# B&R Automation Studio project VisionSample (part 5)

#### Main.st
```iecst
// --------------------------------------------------------------------------------------------------------------------
// This task calculates the nettime depending on a drive velocity
// - This task must run at the same cycle as the Powerlink bus
// - Make sure that nettime is selected in the vision application (Image aquisition -> Aquisition configuration -> Trigger Source -> Trigger delay
// --------------------------------------------------------------------------------------------------------------------
PROGRAM _INIT
	gVisionNettime.CMD.Activate					:= TRUE;
	gVisionNettime.CFG.AxisPeriod				:= 360; // Needs also to be set in the axis configuration
	gVisionNettime.CFG.AxisPositionTrigger		:= 0;
	gVisionNettime.CFG.AxisPositionDelay_Cycles	:= 1; 	// Number of PLK cycles which the axis position is old when it comes to this task (Time from encoder to now in this task)
	gVisionNettime.CFG.VisionPreTrigger_Cycles	:= 4; 	// Number of powerlink cycles the trigger has to be send ahead
														// For camera only 4 is good value, for backlight use 12 with a 800us Powerlink cylce
END_PROGRAM

// -----------------------------------------------------------------------------------------------------------
// Cyclic part
// -----------------------------------------------------------------------------------------------------------
PROGRAM _CYCLIC
	PowerlinkCycle_us			:= NettimeCurrent_us - NettimeLastCycle_us;
	NettimeLastCycle_us			:= NettimeCurrent_us;
	IF gVisionNettime.CMD.Activate AND gVisionNettime.DAT.AxisInVelocity AND gVisionNettime.DAT.AxisVelocity > 0 THEN
		AxisPositionNow			:= gVisionNettime.DAT.AxisPosition + gVisionNettime.DAT.AxisVelocity * PowerlinkCycle_us * gVisionNettime.CFG.AxisPositionDelay_Cycles / 1000000; // When the MpAxis gives us the read position, it is old. So calculate the "now" position
		IF AxisPositionNow > gVisionNettime.CFG.AxisPeriod THEN // modulo correction
			AxisPositionNow		:= AxisPositionNow - gVisionNettime.CFG.AxisPeriod;
		ELSIF AxisPositionNow < 0 THEN // modulo correction
			AxisPositionNow		:= AxisPositionNow + gVisionNettime.CFG.AxisPeriod;
		END_IF
		IF gVisionNettime.DAT.AxisVelocity > 0 THEN
			TriggerPosDelta		:= gVisionNettime.CFG.AxisPositionTrigger - AxisPositionNow;
		ELSE
			TriggerPosDelta		:= AxisPositionNow - gVisionNettime.CFG.AxisPositionTrigger;
		END_IF
		IF TriggerPosDelta < 0 THEN // modulo correction
			TriggerPosDelta		:= TriggerPosDelta + gVisionNettime.CFG.AxisPeriod;
		END_IF
		TriggerTimeDelta_us := LREAL_TO_DINT((TriggerPosDelta / gVisionNettime.DAT.AxisVelocity) * 1000000);
		// Wait for the moment that axis is in the send trigger window depend on delay by topology and the actual powerlink cycle
		IF (TriggerTimeDelta_us >= (gVisionNettime.CFG.VisionPreTrigger_Cycles)     * PowerlinkCycle_us) AND
		   (TriggerTimeDelta_us <= (gVisionNettime.CFG.VisionPreTrigger_Cycles + 1) * PowerlinkCycle_us) THEN
			gVisionNettime.DAT.NettimeNext_us	:= NettimeCurrent_us + TriggerTimeDelta_us;
			gVisionNettime.DAT.NettimeDelta_us	:= TriggerTimeDelta_us;
			// Transfer nettime to sensor and fire trigger
			IF gVisionSensor[gSelectedSensor].HW.Ready AND NOT gVisionSensor[gSelectedSensor].DAT.ImageProcessingActive THEN
				gVisionSensor[gSelectedSensor].CMD.ImageTrigger	:= TRUE;
				gVisionSensor[gSelectedSensor].DAT.NettimeDelay	:= gVisionNettime.DAT.NettimeNext_us;
			ELSE
				gVisionNettime.DAT.Overflow := gVisionNettime.DAT.Overflow + 1;
			END_IF
		END_IF
	END_IF
END_PROGRAM
```

### Program Logical/Vision/Axis (IEC)

#### Main.st - Init, cyclic, exit code
```iecst
// --------------------------------------------------------------------------------------------------------------------
// Motion sample for using nettime
// --------------------------------------------------------------------------------------------------------------------
PROGRAM _INIT
	MpAxisBasic_0.Enable			:= TRUE;
	MpAxisBasic_0.MpLink			:= ADR(gAxis_1);
	MpAxisBasic_0.Parameters		:= ADR(MpAxisBasicPar_0);
	MpAxisBasic_0();
	MpAxisBasicPar_0.Homing.Mode	:= mcHOMING_DEFAULT;
END_PROGRAM

// -----------------------------------------------------------------------------------------------------------
// Cyclic part
// -----------------------------------------------------------------------------------------------------------
PROGRAM _CYCLIC
	MpAxisBasic_0.Power					:= MpAxisBasic_0.Active AND MpAxisBasic_0.Info.ReadyToPowerOn AND cmdAxisPower;
	MpAxisBasic_0.ErrorReset			:= cmdAxisErrorReset;
	MpAxisBasic_0.Home					:= MpAxisBasic_0.PowerOn AND NOT MpAxisBasic_0.IsHomed XOR cmdAxisHome;
	MpAxisBasic_0.MoveVelocity			:= MpAxisBasic_0.PowerOn AND MpAxisBasic_0.IsHomed AND cmdAxisRun;
	IF MpAxisBasic_0.PowerOn AND MpAxisBasic_0.IsHomed AND cmdAxisMoveAbs THEN
		MpAxisBasic_0.MoveAbsolute		:= TRUE;
		MpAxisBasicPar_0.Position		:= gVisionNettime.CFG.AxisPositionTrigger;
	END_IF
	cmdAxisMoveAbs					:= FALSE;
	IF AxisVelocity <> MpAxisBasicPar_0.Velocity OR AxisAcceleration <> MpAxisBasicPar_0.Acceleration THEN
		MpAxisBasicPar_0.Velocity		:= AxisVelocity;
		MpAxisBasicPar_0.Acceleration	:= AxisAcceleration;
		MpAxisBasicPar_0.Deceleration	:= AxisAcceleration;
		MpAxisBasic_0.Update			:= TRUE;
	END_IF
	MpAxisBasic_0();
	gVisionNettime.DAT.AxisInVelocity	:= MpAxisBasic_0.InVelocity;
	gVisionNettime.DAT.AxisPosition		:= MpAxisBasic_0.Position;
	gVisionNettime.DAT.AxisVelocity		:= MpAxisBasic_0.Velocity;
	IF MpAxisBasic_0.UpdateDone THEN
		MpAxisBasic_0.Update := FALSE;
	END_IF
	IF MpAxisBasic_0.InPosition THEN
		MpAxisBasic_0.MoveAbsolute		:= FALSE;
	END_IF
END_PROGRAM
```

#### Variables.var - Local variables
```iecst
VAR
	MpAxisBasicPar_0 : MpAxisBasicParType; (*Motion parameters*)
	MpAxisBasic_0 : MpAxisBasic; (*Basic motion function block*)
	AxisVelocity : REAL := 360; (*Velocity for movement*)
	AxisAcceleration : REAL := 36000; (*Acceleration and deceleration for movement*)
	cmdAxisRun : BOOL;
	cmdAxisPower : BOOL;
	cmdAxisHome : BOOL;
	cmdAxisMoveAbs : BOOL;
	cmdAxisErrorReset : BOOL;
END_VAR
```

#### gAxisTypes.typ - not listed in the package file held
```iecst
(*-----------------------------------------------------------------------------------------------------------------------------------------*)
(*General vision structures*)

TYPE
	gAxis_status_typ : 	STRUCT
		position : REAL;
		velocity : REAL;
		inVelocity : BOOL;
		triggerTimeDelta : DINT;
		nettime : DINT;
		powerlinkCycleTime : DINT;
	END_STRUCT;
	gAxis_typ : 	STRUCT
		status : gAxis_status_typ;
	END_STRUCT;
END_TYPE
```

#### gAxis.var - not listed in the package file held
```iecst
VAR
	gAxis : gAxis_typ;
END_VAR
```

#### Program Logical/Vision/Axis/Axis

##### Variables.var
```iecst
VAR
	this : local_typ;
	hw : hw_typ;
	hmi : hmi_typ;
END_VAR
```

##### Main.st
```iecst
// --------------------------------------------------------------------------------------------------------------------
// Motion sample for using nettime
// --------------------------------------------------------------------------------------------------------------------
PROGRAM _INIT
	this.mpAxisBasic_0.Enable			:= TRUE;
	this.mpAxisBasic_0.MpLink			:= ADR(gAxis_1);
	this.mpAxisBasic_0.Parameters		:= ADR(this.mpAxisBasicPar_0);
	this.mpAxisBasic_0();
	this.mpAxisBasicPar_0.Homing.Mode	:= mcHOMING_DEFAULT;

	gVisionNettime.CMD.Activate					:= TRUE;
	hmi.in.recipe.axisPeriod				:= 360; // Needs also to be set in the axis configuration
	hmi.in.recipe.axisPositionTrigger		:= 0;
	hmi.in.recipe.axisPositionDelayCycles	:= 1; 	// Number of PLK cycles which the axis position is old when it comes to this task (Time from encoder to now in this task)
	hmi.in.recipe.visionPreTriggerCycles	:= 4; 	// Number of powerlink cycles the trigger has to be send ahead
	// For camera only 4 is good value, for backlight use 12 with a 800us Powerlink cylce

END_PROGRAM

// -----------------------------------------------------------------------------------------------------------
// Cyclic part
// -----------------------------------------------------------------------------------------------------------
PROGRAM _CYCLIC

// -----------------------------------------------------------------------------------------------------------
// Mapp Motion Axis control
// -----------------------------------------------------------------------------------------------------------
	this.mpAxisBasic_0.Power				:= this.mpAxisBasic_0.Active AND this.mpAxisBasic_0.Info.ReadyToPowerOn AND hmi.in.cmd.power;
	this.mpAxisBasic_0.ErrorReset			:= hmi.in.cmd.errReset;
	this.mpAxisBasic_0.Home					:= this.mpAxisBasic_0.PowerOn AND NOT this.mpAxisBasic_0.IsHomed XOR hmi.in.cmd.home;
	this.mpAxisBasic_0.MoveVelocity			:= this.mpAxisBasic_0.PowerOn AND this.mpAxisBasic_0.IsHomed AND hmi.in.cmd.run;

	IF this.mpAxisBasic_0.PowerOn AND this.mpAxisBasic_0.IsHomed AND hmi.in.cmd.moveAbs THEN
		this.mpAxisBasic_0.MoveAbsolute		:= TRUE;
		this.mpAxisBasicPar_0.Position		:= gVisionNettime.CFG.AxisPositionTrigger;
	END_IF
	hmi.in.cmd.moveAbs					:= FALSE;

	IF hmi.in.recipe.velocity <> this.mpAxisBasicPar_0.Velocity OR hmi.in.recipe.acceleration <> this.mpAxisBasicPar_0.Acceleration THEN
		this.mpAxisBasicPar_0.Velocity		:= hmi.in.recipe.velocity;
		this.mpAxisBasicPar_0.Acceleration	:= hmi.in.recipe.acceleration;
		this.mpAxisBasicPar_0.Deceleration	:= hmi.in.recipe.acceleration;
		this.mpAxisBasic_0.Update			:= TRUE;
	END_IF

	this.mpAxisBasic_0();

	IF hw.in.nettime > this.nettimeLastCycle_us THEN
		this.powerlinkCycle_us	:= hw.in.nettime - this.nettimeLastCycle_us;
	ELSE
		this.powerlinkCycle_us	:= -2147483648-hw.in.nettime + 2147483647-this.nettimeLastCycle_us; // handle wrap around
	END_IF
	this.nettimeLastCycle_us		:= hw.in.nettime;

	hmi.out.inVelocity 	:= gAxis.status.inVelocity	:= 	this.mpAxisBasic_0.InVelocity;
	hmi.out.veleocity 	:= gAxis.status.velocity	:= 	this.mpAxisBasic_0.Velocity;
	hmi.out.inPostion 								:=	this.mpAxisBasic_0.InPosition;
	// When the MpAxis gives us the read position, it is old. So calculate the "now" position
	hmi.out.positon 	:= gAxis.status.position	:= 	LREAL_TO_REAL(this.mpAxisBasic_0.Position) + this.mpAxisBasic_0.Velocity * DINT_TO_REAL(this.powerlinkCycle_us) * hmi.in.recipe.axisPositionDelayCycles / 1000000; ;

	IF this.mpAxisBasic_0.UpdateDone THEN
		this.mpAxisBasic_0.Update := FALSE;
	END_IF

	IF this.mpAxisBasic_0.InPosition THEN
		this.mpAxisBasic_0.MoveAbsolute		:= FALSE;
	END_IF

	// -----------------------------------------------------------------------------------------------------------
	// Calulate time to camera trigger point
	// -----------------------------------------------------------------------------------------------------------

	// calculate axis postion in the current period
	IF this.axisPositionNow > hmi.in.recipe.axisPeriod THEN // modulo correction
		this.axisPositionNow		:= hmi.out.positon- hmi.in.recipe.axisPeriod;
	ELSIF this.axisPositionNow < 0 THEN // modulo correction
		this.axisPositionNow		:= hmi.out.positon + hmi.in.recipe.axisPeriod;
	END_IF

	// calculate differen (triggerPosDelta) in current axis postion to the trigger postion
	IF this.mpAxisBasic_0.Velocity > 0 THEN
		this.triggerPosDelta		:= hmi.in.recipe.axisPositionTrigger - this.axisPositionNow;
	ELSE
		this.triggerPosDelta		:= this.axisPositionNow - hmi.in.recipe.axisPositionTrigger;
	END_IF

	IF this.triggerPosDelta < 0 THEN // modulo correction
		this.triggerPosDelta		:= this.triggerPosDelta + hmi.in.recipe.axisPositionTrigger;
	END_IF

	IF hmi.out.veleocity > 0 THEN
		// convert position difference to a time difference (the time until the axis is at the trigger postion with the current velocity)
		gAxis.status.triggerTimeDelta 	:= LREAL_TO_DINT((this.triggerPosDelta / this.mpAxisBasic_0.Velocity) * 1000000);
	END_IF

	gAxis.status.nettime 		  		:= hw.in.nettime;
	gAxis.status.powerlinkCycleTime 	:= this.powerlinkCycle_us;

	hmi.out.triggerPosDelta 	:= this.triggerPosDelta;
	hmi.out.powerlinkCycle_us 	:= this.powerlinkCycle_us;
	hmi.out.triggerTimeDelta 	:= this.triggerTimeDelta;

END_PROGRAM
```

### Program Logical/Vision/YourTask (IEC)

#### Types.typ
```iecst
TYPE
	enumViMotion :
		(
		stINIT,
		stPOWER,
		stHOME,
		stREADY,
		stRUN
		);
END_TYPE
```

#### Main.st
```iecst
// -----------------------------------------------------------------------------------------------------------
// Use this task to add your own code
// -----------------------------------------------------------------------------------------------------------

// -----------------------------------------------------------------------------------------------------------
// Initialization
// -----------------------------------------------------------------------------------------------------------
PROGRAM _INIT
END_PROGRAM

// -----------------------------------------------------------------------------------------------------------
// Cyclic part
// -----------------------------------------------------------------------------------------------------------
PROGRAM _CYCLIC
	// -----------------------------------------------------------------------------------------------------------
	// Vision sensor configuration
	// -----------------------------------------------------------------------------------------------------------
	// Configuration for blob
	gVisionSensor[1].CFG.VisionFunction		:= enumBlob;			// Used to run specific code for this vision function
	gVisionSensor[1].CFG.PowerlinkNode		:= 1;					// Powerlink node number
	gVisionSensor[1].CFG.DataStructure		:= ADR(gBlob);			// Global structures that holds all data related to this function
	gVisionSensor[1].CFG.ComponentLink		:= gCameraBlob;			// Vision component name defined under mappVision in the configuration view
	gVisionSensor[1].CFG.ResolutionWidth	:= 1280;
	gVisionSensor[1].CFG.ResolutionHeight	:= 1024;
	// Configuration for code reader
	gVisionSensor[2].CFG.VisionFunction		:= enumCoderReader;
	gVisionSensor[2].CFG.PowerlinkNode		:= 2;
	gVisionSensor[2].CFG.DataStructure		:= ADR(gCodeReader);
	gVisionSensor[2].CFG.ComponentLink		:= gCameraCodeReading;
	gVisionSensor[2].CFG.ResolutionWidth	:= 1280;
	gVisionSensor[2].CFG.ResolutionHeight	:= 1024;
	// Configuration for match
	gVisionSensor[3].CFG.VisionFunction		:= enumMatch;
	gVisionSensor[3].CFG.PowerlinkNode		:= 3;
	gVisionSensor[3].CFG.DataStructure		:= ADR(gMatch);
	gVisionSensor[3].CFG.ComponentLink		:= gCameraMatch;
	gVisionSensor[3].CFG.ResolutionWidth	:= 1280;
	gVisionSensor[3].CFG.ResolutionHeight	:= 1024;
	// Configuration for meaurement
	gVisionSensor[4].CFG.VisionFunction		:= enumMeasurement;
	gVisionSensor[4].CFG.PowerlinkNode		:= 4;
	gVisionSensor[4].CFG.DataStructure		:= ADR(gMT);
	gVisionSensor[4].CFG.ComponentLink		:= gCameraMeasurement;
	gVisionSensor[4].CFG.ResolutionWidth	:= 1280;
	gVisionSensor[4].CFG.ResolutionHeight	:= 1024;
	// Configuration for OCR
	gVisionSensor[5].CFG.VisionFunction		:= enumOCR;
	gVisionSensor[5].CFG.PowerlinkNode		:= 5;
	gVisionSensor[5].CFG.DataStructure		:= ADR(gOCR);
	gVisionSensor[5].CFG.ComponentLink		:= gCameraOCR;
	gVisionSensor[5].CFG.ResolutionWidth	:= 1280;
	gVisionSensor[5].CFG.ResolutionHeight	:= 1024;
	// Configuration for PixelCounter
	gVisionSensor[6].CFG.VisionFunction		:= enumPixelCounter;
	gVisionSensor[6].CFG.PowerlinkNode		:= 6;
	gVisionSensor[6].CFG.DataStructure		:= ADR(gPixel);
	gVisionSensor[6].CFG.ComponentLink		:= gCameraPxl;
	gVisionSensor[6].CFG.ResolutionWidth	:= 1280;
	gVisionSensor[6].CFG.ResolutionHeight	:= 1024;

	// -----------------------------------------------------------------------------------------------------------
	// Lights configuration
	// -----------------------------------------------------------------------------------------------------------
	// Configuration for backlights
	gVisionLight[1].CFG.LightType		:= enumBacklight;
	gVisionLight[1].CFG.PowerlinkNode	:= 10;
	gVisionLight[1].DAT.FlashColor		:= 1;
	gVisionLight[2].CFG.LightType		:= enumBacklight;
	gVisionLight[2].CFG.PowerlinkNode	:= 11;
	gVisionLight[2].DAT.FlashColor		:= 1;
	// Configuration for lightbars
	gVisionLight[3].CFG.LightType		:= enumLightbar;
	gVisionLight[3].CFG.PowerlinkNode	:= 20;
	gVisionLight[3].DAT.FlashColor		:= 1;

	// -----------------------------------------------------------------------------------------------------------
	// Backlight handling, this block can be deleted when no backlights are used
	// -----------------------------------------------------------------------------------------------------------

	// -----------------------------------------------------------------------------------------------------------
	// Trigger selected backlight when selected sensor is triggered
	IF(EDGEPOS(gVisionSensor[gSelectedSensor].CMD.ImageTrigger)) THEN
		gVisionLight[gSelectedLight].DAT.Exposure		:= gVisionSensor[gSelectedSensor].DAT.Exposure;
		gVisionLight[gSelectedLight].DAT.NettimeDelay	:= gVisionSensor[gSelectedSensor].DAT.NettimeDelay;
		gVisionLight[gSelectedLight].CMD.FlashTrigger	:= TRUE;
	END_IF

END_PROGRAM
```

### gFiles.typ
```iecst
TYPE
	gFiles_output_typ : 	STRUCT
		fileDevice : STRING[10];
		ready : BOOL;
	END_STRUCT;
	gFiles_typ : 	STRUCT
		output : gFiles_output_typ;
	END_STRUCT;
END_TYPE
```

### gFiles.var
```iecst
VAR
	gFiles : gFiles_typ;
END_VAR
```

### Program Logical/Vision/Files/Files (IEC)

#### Types.typ
```iecst
TYPE
	local_typ : 	STRUCT
		brdkFileDevUsb : brdkFileDeviceHandler;
		brdkFileDev : brdkFileDeviceHandler;
	END_STRUCT;
END_TYPE
```

#### Variables.var
```iecst
VAR
	this : local_typ;
END_VAR
```

#### Main.st
```iecst
PROGRAM _INIT
	(* Insert code here *)
	this.brdkFileDev.enable := TRUE;
	this.brdkFileDev.setup.plcDrive := F_DRIVE;
	this.brdkFileDev.setup.usbOverrule := FALSE;
	this.brdkFileDev.simulation.pcRootFolder := 'plcSim\MappVisionDemo';
	this.brdkFileDev.simulation.pcHDDrive := C_DRIVE;
	this.brdkFileDev.setup.rootFileDeviceName := 'ROOT_PLC';

	this.brdkFileDev.setup.fileDevices[0].name := 'SIM_BLOB';
	this.brdkFileDev.setup.fileDevices[0].path := 'sim/BLOB';
	this.brdkFileDev.setup.fileDevices[1].name := 'SIM_CR';
	this.brdkFileDev.setup.fileDevices[1].path := 'sim/CR';
	this.brdkFileDev.setup.fileDevices[2].name := 'SIM_MATCH';
	this.brdkFileDev.setup.fileDevices[2].path := 'sim/Match';
	this.brdkFileDev.setup.fileDevices[3].name := 'SIM_MEAS';
	this.brdkFileDev.setup.fileDevices[3].path := 'sim/Measurement';
	this.brdkFileDev.setup.fileDevices[4].name := 'SIM_OCR';
	this.brdkFileDev.setup.fileDevices[4].path := 'sim/OCR';
	this.brdkFileDev.setup.fileDevices[5].name := 'SIM_PXCNT';
	this.brdkFileDev.setup.fileDevices[5].path := 'sim/PxCnt';

	this.brdkFileDevUsb.setup.plcDrive := F_DRIVE;
	this.brdkFileDevUsb.setup.usbOverrule := TRUE;
	this.brdkFileDevUsb.simulation.pcRootFolder := 'plcSim\MappVisionDemo';
	this.brdkFileDevUsb.simulation.pcHDDrive := C_DRIVE;
	this.brdkFileDevUsb.simulation.pcUSBDrive := D_DRIVE;
	this.brdkFileDevUsb.setup.rootFileDeviceName := 'ROOT_USB';

	this.brdkFileDevUsb.setup.fileDevices[0].name := 'IMG';
	this.brdkFileDevUsb.setup.fileDevices[0].path := 'images';
	this.brdkFileDevUsb.setup.fileDevices[1].name := 'RECIPE';
	this.brdkFileDevUsb.setup.fileDevices[1].path := 'Recipe';
	this.brdkFileDevUsb.setup.fileDevices[2].name := 'VI_DIAG';
	this.brdkFileDevUsb.setup.fileDevices[2].path := 'visionDiag';

END_PROGRAM

PROGRAM _CYCLIC
	(* Insert code here *)

	this.brdkFileDev();

	IF EDGEPOS(this.brdkFileDev.ready) THEN
		this.brdkFileDevUsb.enable := TRUE;
	END_IF

	this.brdkFileDevUsb();

	gFiles.output.fileDevice := 'ROOT';
	gFiles.output.ready := this.brdkFileDevUsb.ready;

END_PROGRAM

PROGRAM _EXIT
	(* Insert code here *)

	END_PROGRAM
```

### Program Logical/Vision/Vi_Color (IEC)

#### Main.st - Init, cyclic, exit code
```iecst
PROGRAM _INIT
	// ---------------------------------------------------------------------------------------------------------------------
	// Camera configuration
	gVisionSensor[VI_COLOR_SENSOR].DAT.Gain := 1;
	gVisionSensor[VI_COLOR_SENSOR].DAT.Focus := 14000;
	gVisionSensor[VI_COLOR_SENSOR].DAT.Exposure := 150;
	gVisionSensor[VI_COLOR_SENSOR].DAT.ChromaticLock := TRUE;
	gBlob.EnhancedBlobInformation := TRUE;
	visTableNo;

END_PROGRAM

PROGRAM _CYCLIC
	CASE Step OF
		// ---------------------------------------------------------------------------------------------------------------------
		// Wait for new upload command
		VISTEP_WAIT:
			gVisionColor.DAT.Status := ERR_OK;
			IF gVisionColor.CMD.Evaluate OR gVisionColor.CMD.Teach THEN
				idx := 1;
				brsmemset(ADR(gVisionColor.DAT), 0, SIZEOF(gVisionColor.DAT));
				gVisionColor.CFG.TeachingIndex := visSelectedProduct + 1;
				gVisionColor.DAT.Status := ERR_FUB_BUSY;
				gVisionSensor[VI_COLOR_SENSOR].DAT.Enable := TRUE;
				Step := VISTEP_FLASH;
			END_IF
			// ---------------------------------------------------------------------------------------------------------------------
			// Teach new color
		VISTEP_FLASH:
			// Flash with all available colors
			IF(idx = 1 AND gVisionColor.CFG.FlashColor1 <> 0) THEN
				gVisionSensor[VI_COLOR_SENSOR].DAT.FlashColor := gVisionColor.CFG.FlashColor1;
			ELSIF(idx = 2 AND gVisionColor.CFG.FlashColor2 <> 0) THEN
				gVisionSensor[VI_COLOR_SENSOR].DAT.FlashColor := gVisionColor.CFG.FlashColor2;
			ELSIF(idx = 3 AND gVisionColor.CFG.FlashColor3 <> 0) THEN
				gVisionSensor[VI_COLOR_SENSOR].DAT.FlashColor := gVisionColor.CFG.FlashColor3;
			ELSIF(idx = 4 AND gVisionColor.CFG.FlashColor4 <> 0) THEN
				gVisionSensor[VI_COLOR_SENSOR].DAT.FlashColor := gVisionColor.CFG.FlashColor4;
				// Finish flashing when no color is set
			ELSE
				IF(gVisionColor.CMD.Teach) THEN
					gVisionColor.CMD.Teach := FALSE;
					Step := VISTEP_WAIT;
				ELSE
					Step := VISTEP_CHECK;
				END_IF
				RETURN;
			END_IF
			// Take new image with selected color
			IF NETTIME_ENABLE THEN
				gVisionSensor[VI_COLOR_SENSOR].DAT.NettimeDelay := NettimeCurrent_us + NETTIME_DEFAULT_DELAY;
			END_IF
			gVisionSensor[VI_COLOR_SENSOR].CMD.ImageTrigger 	:= TRUE;
			IF(gVisionColor.CMD.Teach) THEN
				Step := VISTEP_TEACH;
			ELSE
				Step := VISTEP_CHECK;
			END_IF
			// ---------------------------------------------------------------------------------------------------------------------
			// Teach new color
		VISTEP_TEACH:
			// Wait for trigger to finish
			IF(gVisionSensor[VI_COLOR_SENSOR].CMD.ImageTrigger = FALSE) THEN
				IF(gVisionSensor[VI_COLOR_SENSOR].DAT.ResultCnt > 0)  THEN
					IF(idx = 1) THEN
						gVisionColor.CFG.GrayValue1[gVisionColor.CFG.TeachingIndex] := gBlob.MeanGrayValue[1];
					ELSIF(idx = 2) THEN
						gVisionColor.CFG.GrayValue2[gVisionColor.CFG.TeachingIndex] := gBlob.MeanGrayValue[1];
					ELSIF(idx = 3) THEN
						gVisionColor.CFG.GrayValue3[gVisionColor.CFG.TeachingIndex] := gBlob.MeanGrayValue[1];
					ELSIF(idx = 4) THEN
						gVisionColor.CFG.GrayValue4[gVisionColor.CFG.TeachingIndex] := gBlob.MeanGrayValue[1];
					END_IF
					//
					idx := idx + 1;
					IF(idx > 4) THEN
						gVisionColor.CMD.Teach := FALSE;
						Step := VISTEP_WAIT;
					ELSE
						Step := VISTEP_FLASH;
					END_IF
				ELSE
					gVisionColor.DAT.Status := ERR_VI_COLOR_IDENTIFY;
					Step := VISTEP_ERR;
				END_IF
			END_IF
			// ---------------------------------------------------------------------------------------------------------------------
			// Check new product
		VISTEP_CHECK:
			// Wait for trigger to finish
			IF(gVisionSensor[VI_COLOR_SENSOR].CMD.ImageTrigger = FALSE) THEN
				IF(gVisionSensor[VI_COLOR_SENSOR].DAT.ResultCnt > 0)  THEN
					IF(idx = 1) THEN
						gVisionColor.DAT.GrayValue1 := gBlob.MeanGrayValue[1];
					ELSIF(idx = 2) THEN
						gVisionColor.DAT.GrayValue2 := gBlob.MeanGrayValue[1];
					ELSIF(idx = 3) THEN
						gVisionColor.DAT.GrayValue3 := gBlob.MeanGrayValue[1];
					ELSIF(idx = 4) THEN
						gVisionColor.DAT.GrayValue4 := gBlob.MeanGrayValue[1];
					END_IF
					//
					idx := idx + 1;
					IF(idx > 4) THEN
						gVisionColor.DAT.LowError := 16#FFFF;
						gVisionColor.DAT.LowIndex := 16#FFFF;
						gVisionColor.DAT.LowDistance := 16#FFFF;
						Step := VISTEP_EVAL;
					ELSE
						Step := VISTEP_FLASH;
					END_IF
				ELSE
					gVisionColor.DAT.Status := ERR_VI_COLOR_IDENTIFY;
					Step := VISTEP_ERR;
				END_IF
			END_IF
			// ---------------------------------------------------------------------------------------------------------------------
			// Check new product
		VISTEP_EVAL:
			FOR idx:= 1 TO MAX_NUM_PRODUCTS DO
				// Abort when product gray values are empty
				IF(gVisionColor.CFG.GrayValue1[idx] = 0 AND gVisionColor.CFG.GrayValue2[idx] = 0 AND gVisionColor.CFG.GrayValue3[idx] = 0 AND gVisionColor.CFG.GrayValue4[idx] = 0) THEN
					EXIT;
				END_IF
				// Calculate error for all colors and products
				FOR idy:= 1 TO 4 DO
					IF(idy = 1 AND gVisionColor.CFG.FlashColor1 <> 0) THEN
						gVisionColor.DAT.TotalError[idx] := gVisionColor.DAT.TotalError[idx] + ABS(UINT_TO_INT(gVisionColor.DAT.GrayValue1) - gVisionColor.CFG.GrayValue1[idx]);
					ELSIF(idy = 2 AND gVisionColor.CFG.FlashColor2 <> 0) THEN
						gVisionColor.DAT.TotalError[idx] := gVisionColor.DAT.TotalError[idx] + ABS(UINT_TO_INT(gVisionColor.DAT.GrayValue2) - gVisionColor.CFG.GrayValue2[idx]);
					ELSIF(idy = 3 AND gVisionColor.CFG.FlashColor3 <> 0) THEN
						gVisionColor.DAT.TotalError[idx] := gVisionColor.DAT.TotalError[idx] + ABS(UINT_TO_INT(gVisionColor.DAT.GrayValue3) - gVisionColor.CFG.GrayValue3[idx]);
					ELSIF(idy = 4 AND gVisionColor.CFG.FlashColor4 <> 0) THEN
						gVisionColor.DAT.TotalError[idx] := gVisionColor.DAT.TotalError[idx] + ABS(UINT_TO_INT(gVisionColor.DAT.GrayValue4) - gVisionColor.CFG.GrayValue4[idx]);
					END_IF
				END_FOR;
				// New lowest error
				IF(gVisionColor.DAT.TotalError[idx] < gVisionColor.DAT.LowError) THEN
					gVisionColor.DAT.LowError := gVisionColor.DAT.TotalError[idx];
					gVisionColor.DAT.LowIndex := idx;
					gVisionColor.DAT.LowName := gVisionColor.CFG.ProductName[idx];
				END_IF
			END_FOR;
			// Check distance to next best value
			IF(gVisionColor.DAT.LowIndex <> 16#FFFF) THEN
				FOR idx:= 1 TO MAX_NUM_PRODUCTS DO
					// Abort when product gray values are empty
					IF(gVisionColor.CFG.GrayValue1[idx] = 0 AND gVisionColor.CFG.GrayValue2[idx] = 0 AND gVisionColor.CFG.GrayValue3[idx] = 0 AND gVisionColor.CFG.GrayValue4[idx] = 0) THEN
						EXIT;
					END_IF
					// Store next best product
					IF(gVisionColor.DAT.LowIndex <> idx AND INT_TO_UINT(ABS(UINT_TO_INT(gVisionColor.DAT.TotalError[gVisionColor.DAT.LowIndex])) - gVisionColor.DAT.TotalError[idx]) < gVisionColor.DAT.LowDistance) THEN
						gVisionColor.DAT.LowDistance := ABS(UINT_TO_INT(gVisionColor.DAT.TotalError[gVisionColor.DAT.LowIndex]) - gVisionColor.DAT.TotalError[idx]);
					END_IF
				END_FOR;
				visSelectedProduct := gVisionColor.DAT.LowIndex - 1;
			END_IF
			// Make sure we dont exceed max error
			IF(gVisionColor.DAT.LowError > gVisionColor.CFG.MaxError) THEN
				gVisionColor.DAT.Status := ERR_VI_COLOR_MAX_ERROR;
				Step := VISTEP_ERR;
				// Make sure we have enough distance to next best value
			ELSIF(gVisionColor.DAT.LowDistance < gVisionColor.CFG.MinDifference) THEN
				gVisionColor.DAT.Status := ERR_VI_COLOR_MIN_DISTANCE;
				Step := VISTEP_ERR;
				// Make sure we dont exceed max error
			ELSE
				gVisionColor.CMD.Evaluate := FALSE;
				Step := VISTEP_WAIT;
			END_IF
			// ---------------------------------------------------------------------------------------------------------------------
			// Error state
		VISTEP_ERR:
			IF gVisionColor.CMD.ResetError THEN
				gVisionColor.CMD.ResetError := FALSE;
				gVisionColor.DAT.Status := 0;
				Step := VISTEP_WAIT;
			ELSE
				brsmemset(ADR(gVisionColor.CMD), 0, SIZEOF(gVisionColor.CMD));
			END_IF
	END_CASE
END_PROGRAM
```

#### Variables.var - Local variables
```iecst
(*-----------------------------------------------------------------------------------------------------------------------------------------*)
(*Local variables*)
VAR
	Step : VIStep_Enum;
	idy : UINT;
	idx : UINT;
	visSelectedProduct : UINT;
	visTableNo : ARRAY[1..MAX_NUM_PRODUCTS] OF USINT := [1,2,3,4,5,6,7,8];
END_VAR
(*-----------------------------------------------------------------------------------------------------------------------------------------*)
(*Local constants*)
VAR CONSTANT
	VI_COLOR_SENSOR : USINT := 1; (*Camera index used for color detection*)
END_VAR
(*-----------------------------------------------------------------------------------------------------------------------------------------*)
(*Error contants*)
VAR CONSTANT
	ERR_VI_COLOR_IDENTIFY : UINT := 10000; (*No result found*)
	ERR_VI_COLOR_MAX_ERROR : UINT := 10001; (*Error exceeds maximum value*)
	ERR_VI_COLOR_MIN_DISTANCE : UINT := 10002; (*Next best value is too close*)
END_VAR
```

### Program Logical/Vision/Vi_light

#### Variables.var
```iecst
(*-----------------------------------------------------------------------------------------------------------------------------------------*)
VAR
	VisionLight : REFERENCE TO typLightMain; (*General vision functions that are independent from the inspection function*)
	FlashFailedCntOld : ARRAY[1..MAX_NUM_LIGHTS] OF USINT;
	FlashCompletedCntOld : ARRAY[1..MAX_NUM_LIGHTS] OF USINT;
	visLightsTrigger : BOOL;
	visLightsReset : BOOL;
	visEnableCommand : BOOL;
	visSelectedFlashColor : STRING[10]; (*Flash color string*)
	TriggerTimeout : ARRAY[1..MAX_NUM_LIGHTS] OF TON; (*Disable web reload when timed out*)
	InitialSearchLight : BOOL;
	i : INT;
	visSelectedFlashColorOld : STRING[10];
	visEnableLightBarValues : BOOL;
	idx : UINT;
END_VAR
```

#### Main.st
```iecst
// --------------------------------------------------------------------------------------------------------------------
// General external lights task. This is a support task for the mappView visualization.
// Version 1.x (Check revision history for details)
// --------------------------------------------------------------------------------------------------------------------
PROGRAM _INIT
	// Map global structure to local reference
	VisionLight ACCESS ADR(gVisionLight[visSelectedLight]);

	InitialSearchLight := TRUE;
END_PROGRAM

// -----------------------------------------------------------------------------------------------------------
// Cyclic part
// -----------------------------------------------------------------------------------------------------------
PROGRAM _CYCLIC
// -----------------------------------------------------------------------------------------------------------
// Part 1: Things to be done for every light
// -----------------------------------------------------------------------------------------------------------
	FOR idx := 1 TO MAX_NUM_LIGHTS DO
		// -----------------------------------------------------------------------------------------------------------
		// Reset Light trigger
		// -----------------------------------------------------------------------------------------------------------
		IF (gVisionLight[idx].DAT.FlashCompletedCnt <> FlashCompletedCntOld[idx] OR gVisionLight[idx].DAT.FlashFailedCnt <> FlashFailedCntOld[idx]) THEN
			FlashCompletedCntOld[idx]			:= gVisionLight[idx].DAT.FlashCompletedCnt;
			FlashFailedCntOld[idx]				:= gVisionLight[idx].DAT.FlashFailedCnt;
			gVisionLight[idx].CMD.FlashTrigger	:= FALSE;
		END_IF

		// -----------------------------------------------------------------------------------------------------------
		// Reset trigger when timed out
		// -----------------------------------------------------------------------------------------------------------
		IF gVisionLight[idx].CMD.FlashTrigger THEN
			TriggerTimeout[idx].IN := TRUE;
			TriggerTimeout[idx].PT := REAL_TO_TIME(gVisionLight[idx].DAT.Timeout * 1.25);
			IF TriggerTimeout[idx].Q THEN
				gVisionLight[idx].CMD.FlashTrigger		:= FALSE;
				gVisionLight[idx].CMD.FlashTriggerReset	:= TRUE;
			END_IF
		ELSE
			TriggerTimeout[idx].IN := FALSE;
			gVisionLight[idx].CMD.FlashTriggerReset := FALSE;
		END_IF
		TriggerTimeout[idx]();
	END_FOR

// -----------------------------------------------------------------------------------------------------------
// Part 2: Things to be done for the actual selected light / visualization related things
// -----------------------------------------------------------------------------------------------------------
	// -----------------------------------------------------------------------------------------------------------
	// Select first available light after reboot
	// -----------------------------------------------------------------------------------------------------------
	IF InitialSearchLight THEN
		FOR i := 1 TO MAX_NUM_LIGHTS DO
			IF gVisionLight[i].HW.Connected THEN
				visSelectedLight := i;
				InitialSearchLight := FALSE;
				EXIT;
			END_IF
		END_FOR
	END_IF
	 // -----------------------------------------------------------------------------------------------------------
	// Map global structure to local reference
	// -----------------------------------------------------------------------------------------------------------
	// Make sure we dont exceed array limit
	IF(visSelectedLight > MAX_NUM_LIGHTS) THEN
		visSelectedLight := 1;
	END_IF
	IF(visSelectedLight < 1) THEN
		visSelectedLight := MAX_NUM_LIGHTS;
	END_IF
	VisionLight ACCESS ADR(gVisionLight[visSelectedLight]);

	// -----------------------------------------------------------------------------------------------------------
	// Translate flash color from mappView to IO mapping
	// -----------------------------------------------------------------------------------------------------------
	// Hint: Normally copy from recipe (VisionLight) to visu. Only in case of a change in the visu copy to recipe
	IF visSelectedFlashColor <> visSelectedFlashColorOld THEN // The flash color was changed in the mappView visualization
		VisionLight.DAT.FlashColor := UDINT_TO_USINT(brsatoi(ADR(visSelectedFlashColor)));
	ELSE
		brsitoa(VisionLight.DAT.FlashColor, ADR(visSelectedFlashColor));
	END_IF
	visSelectedFlashColorOld := visSelectedFlashColor;

	// -----------------------------------------------------------------------------------------------------------
	// Reset Light trigger manually
	// -----------------------------------------------------------------------------------------------------------
	IF (visLightsReset) THEN
		VisionLight.CMD.FlashTrigger := FALSE;
		visLightsReset := FALSE;
	END_IF

	// -----------------------------------------------------------------------------------------------------------
	// Fire trigger for lights
	// -----------------------------------------------------------------------------------------------------------
	IF(visLightsTrigger AND VisionLight.HW.Ready) THEN
		// Add default delay and fire trigger
		VisionLight.DAT.NettimeDelay := NettimeCurrent_us + NETTIME_DEFAULT_DELAY;
		VisionLight.CMD.FlashTrigger := TRUE;
		visLightsTrigger := FALSE;
	END_IF

	// -----------------------------------------------------------------------------------------------------------
	// Disable command button when light is disconnected or not ready
	// -----------------------------------------------------------------------------------------------------------
	IF(NOT VisionLight.HW.Connected OR NOT VisionLight.HW.Ready) THEN
		visEnableCommand := FALSE;
	ELSE
		visEnableCommand := TRUE;
	END_IF

	// -----------------------------------------------------------------------------------------------------------
	// Enable fields for different light types
	// -----------------------------------------------------------------------------------------------------------
	visEnableLightBarValues := VisionLight.CFG.LightType = enumLightbar;
END_PROGRAM
```

### Program Logical/Vision/Vi_Optics (IEC)

#### Main.st
```iecst
PROGRAM _INIT

END_PROGRAM
PROGRAM _CYCLIC
	CASE ReadStep OF // Use AsIODiag library to search the ordnernumber of the selcted/plugged camera (eg. VSS112Q22.041P-000) to get the lens and sensor information
		0: // Wait
			IF cmdReadCameraInfo THEN
				cmdReadCameraInfo			:= FALSE;
				Index						:= 0;
				OrderNr						:= '';
				ReadStep := 1;
			END_IF
		1: // Create DiagInformation
			DiagCreateInfo_0.enable			:= TRUE;
			DiagCreateInfo_0.infoKind		:= asdiagPLUGGED;
			DiagCreateInfo_0();
			IF DiagCreateInfo_0.status = 0 THEN
				ReadStep := 2;
			ELSIF DiagCreateInfo_0.status <> ERR_FUB_BUSY THEN
				ReadStep := 90;
			END_IF
		2: // Read HW-ID and compare with selected camera
			DiagGetNumInfo_0.enable			:= TRUE;
			DiagGetNumInfo_0.ident			:= DiagCreateInfo_0.ident;
			DiagGetNumInfo_0.index			:= Index;
			DiagGetNumInfo_0.infoCode		:= asdiagPLUGGED_MODNO;
			DiagGetNumInfo_0();
			IF DiagGetNumInfo_0.status = 0 THEN
				IF DiagGetNumInfo_0.value = gVisionSensor[visSelectedSensor].HW.ID THEN
					ReadStep := 3;
				ELSE
					Index := Index + 1;
					IF Index >= DiagCreateInfo_0.nrEntries THEN
						ReadStep := 91;
					END_IF
				END_IF
			ELSIF DiagGetNumInfo_0.status <> ERR_FUB_BUSY THEN
				ReadStep					:= 92;
			END_IF
		3: // Read ordernumber
			DiagGetStrInfo_0.enable			:= TRUE;
			DiagGetStrInfo_0.ident			:= DiagCreateInfo_0.ident;
			DiagGetStrInfo_0.index			:= Index;
			DiagGetStrInfo_0.infoCode		:= asdiagPLUGGED_MODULE; // Ordnernumber of the plugged module (eg. VSS112Q22.041P-000)
			DiagGetStrInfo_0.pBuffer		:= ADR(OrderNr);
			DiagGetStrInfo_0.bufferLen		:= SIZEOF(OrderNr) - 1;
			DiagGetStrInfo_0();
			IF DiagGetStrInfo_0.status = 0 THEN
				ReadStep := 10;
			ELSIF DiagGetStrInfo_0.status <> ERR_FUB_BUSY THEN
				ReadStep := 93;
			END_IF
		10:
			DiagDisposeInfo_0.enable		:= TRUE;
			DiagDisposeInfo_0.ident			:= DiagCreateInfo_0.ident;
			DiagDisposeInfo_0();
			IF DiagDisposeInfo_0.status = 0 THEN
				ReadStep := 20;
			ELSIF DiagDisposeInfo_0.status <> ERR_FUB_BUSY THEN
				ReadStep := 94;
			END_IF
		20: // get the info to the actual camara, e.g. VSS112Q22.041P-000
			IF brsstrlen(ADR(OrderNr)) = 18 THEN
				pChar ACCESS ADR(OrderNr) + 8; // Letter for Sensor
				CASE pChar OF
					16#31:  Sensor := SENSOR_1_3_MP; // ASCII '1'
					16#32:  Sensor := SENSOR_1_3_MP; // ASCII '2'
					16#34:  Sensor := SENSOR_3_5_MP; // ASCII '4'
					16#35:  Sensor := SENSOR_5_3_MP; // ASCII '5'
				ELSE
					ReadStep := 95;
				END_CASE
				pChar ACCESS ADR(OrderNr) + 10; // first letter for optics (0 or M)
				CASE pChar OF
					16#30:  Lens := LENS_4_6; // ASCII '0'
					16#4D:  Lens := LENS_12_0_MACRO; // ASCII 'M'
				ELSE
					ReadStep := 96;
				END_CASE
				pChar ACCESS ADR(OrderNr) + 11; // second letter for optics
				CASE pChar OF
					16#30:  Lens := LENS_4_6; // ASCII '0' // no optics
					16#32:  Lens := LENS_4_6; // ASCII '2'
					16#33:  Lens := LENS_6_0; // ASCII '3'
					16#34:  Lens := LENS_8_0; // ASCII '4'
					16#35: // ASCII '5'
						IF Lens = LENS_12_0_MACRO THEN
							// do noting, already selected
						ELSE
							Lens := LENS_12_0;
						END_IF
					16#36:  Lens := LENS_16_0; // ASCII '6'
					16#37:  Lens := LENS_25_0; // ASCII '7'
				ELSE
					ReadStep := 97;
				END_CASE
				Distance_mm	:= UINT_TO_LREAL(gVisionSensor[visSelectedSensor].DAT.Focus) / 100.0;
				ReadStep := 0;
			ELSE
				ReadStep := 98;
			END_IF
		90..99: // auto reset errors
			ReadStep := 0;
	END_CASE

	CASE Sensor OF
		SENSOR_1_3_MP:
			PixelSize_um		:= 4.8;
			ResolutionX			:= 1280;
			ResolutionY			:= 1024;
		SENSOR_3_5_MP:
			PixelSize_um		:= 3.2;
			ResolutionX			:= 2112;
			ResolutionY			:= 1664;
		SENSOR_5_3_MP:
			PixelSize_um		:= 3.2;
			ResolutionX			:= 2592;
			ResolutionY			:= 2048;
	END_CASE
	CASE Lens OF
		LENS_4_6:
			FocalLength_mm		:= 4.6;
			MinObjectDist_mm	:= 25;
			MaxObjectDist_mm	:= 65550;
			Aperture			:= 3.5;
		LENS_6_0:
			FocalLength_mm		:= 6.0;
			MinObjectDist_mm	:= 50;
			MaxObjectDist_mm	:= 65550;
			Aperture			:= 3.5;
		LENS_8_0:
			FocalLength_mm		:= 8.0;
			MinObjectDist_mm	:= 50;
			MaxObjectDist_mm	:= 65500;
			Aperture			:= 3.5;
		LENS_12_0:
			FocalLength_mm		:= 12.0;
			MinObjectDist_mm	:= 75;
			MaxObjectDist_mm	:= 5000;
			Aperture			:= 4.0;
		LENS_16_0:
			FocalLength_mm		:= 16.0;
			MinObjectDist_mm	:= 100;
			MaxObjectDist_mm	:= 1500;
			Aperture			:= 4.0;
		LENS_25_0:
			FocalLength_mm		:= 25.0;
			MinObjectDist_mm	:= 250;
			MaxObjectDist_mm	:= 1500;
			Aperture			:= 4.0;
		LENS_12_0_MACRO:
			FocalLength_mm		:= 12.0;
			MinObjectDist_mm	:= 35;
			MaxObjectDist_mm	:= 65;
			Aperture			:= 4.0;
	END_CASE
	ValidDistance					:= Distance_mm >= MinObjectDist_mm AND Distance_mm <= MaxObjectDist_mm;
	IF ValidDistance THEN
		DistanceLens_mm				:= Distance_mm + DISTANCE_FRONTGLASS_LENS_MM; // The lens is 15mm behind the front glass
		IF Binning THEN
			PixelSizeBinning_um		:= PixelSize_um * 2;
		ELSE
			PixelSizeBinning_um		:= PixelSize_um * 1;
		END_IF
		CircleOfConfusion_mm		:= PixelSizeBinning_um * 1 * SQRT(2.0) / 1000.0;
		HyperFocalDistance_mm		:= (FocalLength_mm * FocalLength_mm) / (Aperture * CircleOfConfusion_mm ) + FocalLength_mm;
	    DepthOfFieldNearPos_mm		:= DistanceLens_mm * (HyperFocalDistance_mm - FocalLength_mm) / (HyperFocalDistance_mm + DistanceLens_mm - 2 * FocalLength_mm) - DISTANCE_FRONTGLASS_LENS_MM;
		IF DistanceLens_mm < HyperFocalDistance_mm THEN
			DepthOfFieldFarPos_mm	:= DistanceLens_mm * (HyperFocalDistance_mm - FocalLength_mm) / (HyperFocalDistance_mm - DistanceLens_mm) - DISTANCE_FRONTGLASS_LENS_MM;
			DepthOfField_mm			:= DepthOfFieldFarPos_mm - DepthOfFieldNearPos_mm;
		ELSE
			DepthOfFieldFarPos_mm	:= -1; // Means "infinite"
			DepthOfField_mm			:= -1; // Means "infinite"
		END_IF
		FieldOfView_X_mm			:= PixelSizeBinning_um / 1000 * ResolutionX *(DistanceLens_mm / FocalLength_mm - 1.0);
		FieldOfView_Y_mm			:= PixelSizeBinning_um / 1000 * ResolutionY *(DistanceLens_mm / FocalLength_mm - 1.0);
		Resolution_mmPerPx			:= FieldOfView_X_mm / ResolutionX;
	ELSE
		DistanceLens_mm				:= 0;
		PixelSizeBinning_um			:= 0;
		CircleOfConfusion_mm		:= 0;
		HyperFocalDistance_mm		:= 0;
	    DepthOfFieldNearPos_mm		:= 0;
		DepthOfFieldFarPos_mm		:= 0;
		DepthOfField_mm				:= 0;
		FieldOfView_X_mm			:= 0;
		FieldOfView_Y_mm			:= 0;
		Resolution_mmPerPx			:= 0;
	END_IF
END_PROGRAM
```

#### Variables.var
```iecst
(*Read camera ordernumber*)
VAR
	cmdReadCameraInfo : BOOL;
	DiagCreateInfo_0 : DiagCreateInfo;
	DiagGetNumInfo_0 : DiagGetNumInfo;
	DiagGetStrInfo_0 : DiagGetStrInfo;
	DiagDisposeInfo_0 : DiagDisposeInfo;
	OrderNr : STRING[80];
	ReadStep : INT;
	Index : UDINT;
	pChar : REFERENCE TO USINT;
END_VAR
(**)
(*Inputs*)
VAR
	Distance_mm : LREAL; (*Distance object to camera front glass*)
	Sensor : USINT;
	Lens : USINT;
	Binning : BOOL;
END_VAR
(**)
(*Sensor and lens depending values*)
VAR
	PixelSize_um : LREAL;
	ResolutionX : INT;
	ResolutionY : INT;
	FocalLength_mm : LREAL;
	MinObjectDist_mm : LREAL;
	MaxObjectDist_mm : LREAL;
	Aperture : LREAL;
END_VAR
(**)
(*Internal*)
VAR
	DistanceLens_mm : LREAL;
	PixelSizeBinning_um : LREAL;
	CircleOfConfusion_mm : LREAL;
	HyperFocalDistance_mm : LREAL;
END_VAR
(**)
(*Outputs (calculated)*)
VAR
	ValidDistance : BOOL;
	DepthOfFieldNearPos_mm : LREAL;
	DepthOfFieldFarPos_mm : LREAL;
	DepthOfField_mm : LREAL;
	FieldOfView_X_mm : LREAL;
	FieldOfView_Y_mm : LREAL;
	Resolution_mmPerPx : LREAL;
END_VAR
(**)
(*Constants*)
VAR CONSTANT
	DISTANCE_FRONTGLASS_LENS_MM : LREAL := 15.0;
	SENSOR_1_3_MP : USINT := 0;
	SENSOR_3_5_MP : USINT := 1;
	SENSOR_5_3_MP : USINT := 2;
	LENS_4_6 : USINT := 0;
	LENS_6_0 : USINT := 1;
	LENS_8_0 : USINT := 2;
	LENS_12_0 : USINT := 3;
	LENS_16_0 : USINT := 4;
	LENS_25_0 : USINT := 5;
	LENS_12_0_MACRO : USINT := 6;
END_VAR
```

- Vision Demo Application.docx (binary file, 3234942 bytes)
- Visualisation Logical/mappView (not shown)

- Project.language (not shown)

### RecVariables.var
```iecst
(*------------------------------------------------------------------------------------------------------------------------------------------------------------------------------------------------------------------------*)
(*Configuration for recipe managment*)
VAR CONSTANT
	REC_USE_UNICODE : BOOL := FALSE; (*Use standard strings for recipe name when false, use unicode strings for recipe name when true*)
	REC_SORT_NUMERIC : BOOL := FALSE; (*Sort recipe names as numeric values instead of alphabetic*)
	REC_RECIPE_TYPE : recTYPE := typeCSV; (*Type of recipe (CSV / XML)*)
END_VAR
VAR
	REC_MPLINK : {REDUND_UNREPLICABLE} STRING[80] := 'gRecipeCsv_01'; (*mappRecipe link name from configuration view. User gRecipeCsv_01 for CSV and gRecipeXml_01 for XML in this demo*)
END_VAR
VAR CONSTANT
	REC_DEVICE : STRING[80] := 'VisionFileDevice'; (*Device name for the recipe data defined under File Devices in the CPU configuration*)
	REC_DIRECTORY : STRING[80] := 'Recipe_01'; (*Directory where the recipes are stored*)
	REC_THIS_TASK : STRING[40] := 'Recipe_01'; (*Name of this task and the global variables structure*)
	REC_REC_NUM : USINT := 100; (*Maximum number of recipes*)
	REC_VAR_NUM : USINT := 10; (*Maximum number of variables that can be registered*)
	REC_NAME_LENGTH : USINT := 40; (*Maximum length for a recipe name*)
	REC_UPLOAD_DOWNLOAD_SIZE : UDINT := 100000; (*Maximum size of memory allocated for uploading and downloading files*)
	REC_VIS_LENGTH : USINT := 120; (*Make this REC_NAME_LENGTH  x3*)
	REC_MAX_CLIENTS_ID : USINT := 2; (*Highest client ID for concurrent web client connections. Do not change this number.*)
END_VAR
VAR
	REC_VIEW_FILTER : ARRAY[0..9] OF STRING[5] := ['csv','xml',8('')]; (*Files extensions than can be used with the view command*)
END_VAR
(*------------------------------------------------------------------------------------------------------------------------------------------------------------------------------------------------------------------------*)
(*Add you variables to this list*)
VAR
	REC_VAR_LIST : ARRAY[1..REC_VAR_NUM] OF STRING[100] := ['RecipeData','','','','','','','',2('')]; (*List of variables to be inlcuded in a recipe*)
	Recipe_01 : recMAIN; (*Global recipe structure. The name must match the task name of the recipe managment.*)
END_VAR
```

### Program Logical/mappRecipe/Recipe_01 (IEC)

#### Init.st - Init and local configuration
```iecst
// --------------------------------------------------------------------------------------------------------------------
//	Function:	Recipe management with mappRecipe
//  Version:	0.7
//	Changed:	08.05.2020
// --------------------------------------------------------------------------------------------------------------------

PROGRAM _INIT
	// ----------------------------------------------------------------------------------------
	// The following settings can be adjusted
	IF(DiagCpuIsSimulated()) THEN
		DeviceName 	:= 'SIM_DEVICE';						// Device name from the CPU configuration for simulation
	ELSE
		DeviceName 	:= REC_DEVICE;							// Device name from the CPU configuration for X20CPU
	END_IF

	// ----------------------------------------------------------------------------------------
	// Dont change anything below this line
	// ----------------------------------------------------------------------------------------

	// ----------------------------------------------------------------------------------------
	// Make sure global variable structure and task name are correct
	taskStatus := ST_ident(ADR(REC_THIS_TASK), taskGroup, ADR(taskID));
	pvStatus := PV_xgetadr(ADR(REC_THIS_TASK), ADR(pvADR), ADR(pvLEN));
	// Connect global and local structure
	IF(pvStatus = 0) THEN
		RECIPE ACCESS pvADR;
		brsmemset(ADR(RECIPE.ERR), 0 , SIZEOF(RECIPE.ERR));
		RECIPE.PAR.Initialized := FALSE;
	END_IF

	// ----------------------------------------------------------------------------------------
	// Get mapp link information
	MpComGetLink_0.Enable := TRUE;
	MpComGetLink_0.ComponentName := ADR(REC_MPLINK);
	MpComGetLink_0();
	// Create error
	IF(MpComGetLink_0.Error) THEN
		rec_state := CreateError(ADR(RECIPE), ERR_REC_MPLINK, "mplink name is incorrect", rec_state);
	END_IF

	// ----------------------------------------------------------------------------------------
	// Allocate memory for file upload and download
	AsMemPartCreate_0.enable	:= TRUE;
	AsMemPartCreate_0.len		:= REC_UPLOAD_DOWNLOAD_SIZE;
	AsMemPartCreate_0();
	IF AsMemPartCreate_0.status <> 0 THEN
		rec_state := CreateError(ADR(RECIPE), ERR_MEM_ALLOC, "file upload and download memory alloc failed", rec_state);
	ELSE
		AsMemPartAllocClear_0.enable	:= TRUE;
		AsMemPartAllocClear_0.ident		:= AsMemPartCreate_0.ident;
		AsMemPartAllocClear_0.len		:= REC_UPLOAD_DOWNLOAD_SIZE;
		AsMemPartAllocClear_0();
		IF AsMemPartAllocClear_0.status <> 0 THEN
			rec_state := CreateError(ADR(RECIPE), ERR_MEM_ALLOC, "file upload and download memory clear failed", rec_state);
		END_IF
	END_IF

	// ----------------------------------------------------------------------------------------
	// Generate HTML messages for web upload
	upload_response	:= '<html><body><form action="/uploadA.html" name="form_upload" method="post" enctype="multipart/form-data" >
	<label for="file-upload" style="font-weight:bold;font-family: sans-serif;font-size:16px;padding:15px 50px;10px;10px;" class="custom-file-upload">Upload</label>
	<input type="file" id="file-upload" style="display:none;" onchange="form.submit()" name="file_selected" content-type="application/octet-stream" />
	</form><body></html> ';
	WebServiceUpload.pServiceName := ADR('uploadA.html');
END_PROGRAM
```
